ABB RobotStudio station: Romantici.rspag

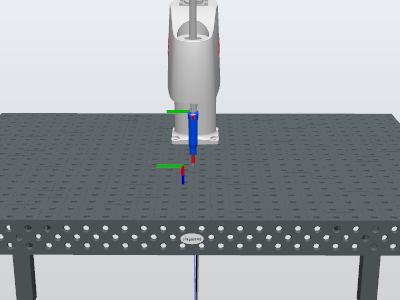
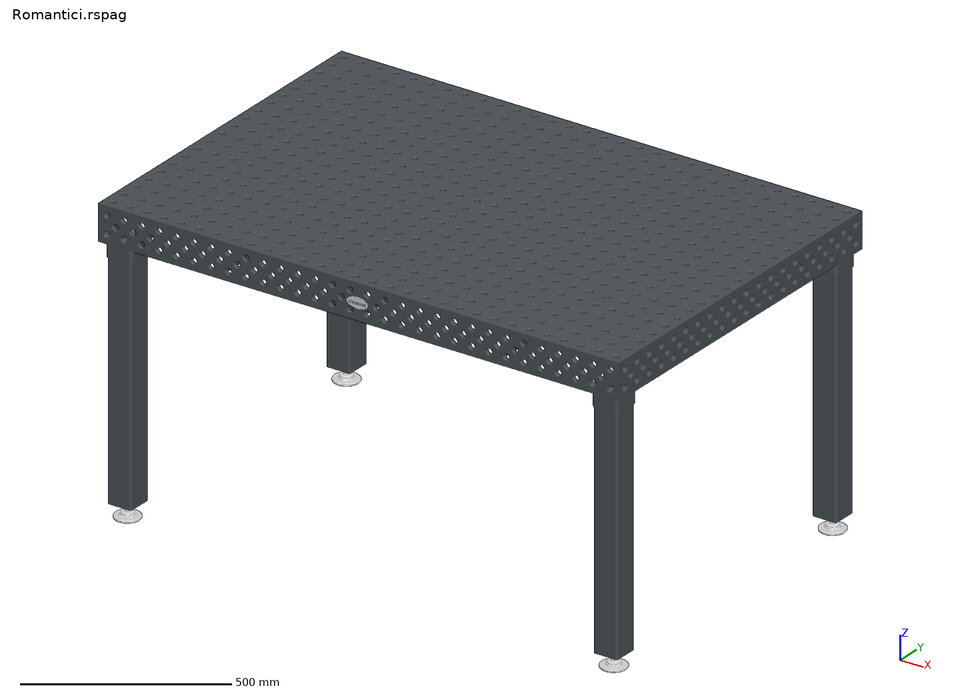
[picture v1: parts stored in the station drawn from their meshes, with robot base, taught points and paths (robot models come from the ABB library and are not in the file)]
Station Solution_1_Tutorial (saved by RobotStudio 22.3.10190.2)
Layout (positions relative to the parent item):
  - table [part] at (-200, -500, 830) mm
  - siegmund_1500_1000 [part], size 1500 x 1010.3 x 830 mm
  - IRB910SC_3_45__01 [mechanism, from Robots\IRB910SC_3_45__01.rslib] at (0, 200, 830) mm, rotated rx 0 ry 0 rz -90 deg; joint values [0, 0, 0, 0] (rad or m)
  - PencilHolder [mechanism] at (0, -250, 1050.2) mm, rotated rx 180 ry 0 rz 0 deg
      TCP PencilHolder at (-72.46, -108.4, 17) mm, rotated rx 90 ry 0 rz 0 deg
      links: Assembly3
  - Rámec_1 [frame] at (0, 30, 162.64) mm
Attachment: PencilHolder is attached to IRB910SC_3_45__01 / Link4
Targets, tools, work objects and paths stored in the station, written as RAPID:
! task (no controller)
MODULE CalibData
  PERS tooldata PencilHolder:=[TRUE,[[0,30,162.643],[1,0,0,0]],[1,[0,0,1],[1,0,0,0],0,0,0]];
ENDMODULE

